(* IEC 61131-3 sources: Word/plc-course/10-structured-text/labs/solutions, 4 files *)

(* ---- 10-1-array-statistics.st ---- *)
(* Lab 10-1: Array statistics - ten cold-store temperature probes.
   Module 10 (Structured Text). REFERENCE SOLUTION - try the lab yourself first. *)

PROGRAM ArrayStats
  VAR (* interface: the I/O mapping routine copies the ten probe readings in here *)
    Samples  : ARRAY[1..10] OF REAL;  (* probe temperatures, degC. Samples[3] is probe TT-303 *)
    MinValue : REAL;                  (* coldest reading, degC *)
    MaxValue : REAL;                  (* warmest reading, degC *)
    Average  : REAL;                  (* mean of the ten readings, degC *)
    MaxIndex : INT;                   (* probe number (1..10) of the warmest reading *)
  END_VAR
  VAR CONSTANT
    NUM_PROBES : INT := 10;           (* must match the upper bound of Samples *)
  END_VAR
  VAR
    i   : INT;                        (* loop index *)
    Sum : REAL;                       (* running total, rebuilt from zero every scan *)
  END_VAR

  (* Start from the first sample, never from 0.0. In a freezer every reading is
     below zero, so a maximum that started at 0.0 would never be beaten. *)
  MinValue := Samples[1];
  MaxValue := Samples[1];
  MaxIndex := 1;
  Sum := 0.0;   (* Sum keeps its value between scans, so it must be cleared here *)

  FOR i := 1 TO NUM_PROBES DO
    Sum := Sum + Samples[i];

    IF Samples[i] < MinValue THEN
      MinValue := Samples[i];
    END_IF;

    (* Strictly greater: when two probes share the warmest value, the
       first one found (the lower probe number) is kept. *)
    IF Samples[i] > MaxValue THEN
      MaxValue := Samples[i];
      MaxIndex := i;
    END_IF;
  END_FOR;

  (* REAL division: both operands must be REAL, so convert the count. *)
  Average := Sum / INT_TO_REAL(NUM_PROBES);
END_PROGRAM

CONFIGURATION Config0
  RESOURCE Res0 ON PLC
    TASK MainTask(INTERVAL := T#10ms, PRIORITY := 0);
    PROGRAM Inst0 WITH MainTask : ArrayStats;
  END_RESOURCE
END_CONFIGURATION

(* ---- 10-2-median-filter.st ---- *)
(* Lab 10-2: Median filter for a noisy tank level.
   Module 10 (Structured Text). REFERENCE SOLUTION - try the lab yourself first. *)

PROGRAM MedianFilter
  VAR (* interface *)
    RawLevel      : REAL;   (* noisy level from the radar transmitter, % *)
    SampleTrig    : BOOL;   (* sample clock: each rising edge takes one sample *)
    FilteredLevel : REAL;   (* median of the last five samples, % *)
    Ready         : BOOL;   (* TRUE once five samples have been collected *)
  END_VAR
  VAR
    History    : ARRAY[1..5] OF REAL;  (* samples in arrival order: [1] oldest, [5] newest *)
    Sorted     : ARRAY[1..5] OF REAL;  (* working copy that gets sorted *)
    Count      : INT;                  (* samples collected so far, 0..5 *)
    SampleEdge : R_TRIG;               (* one sample per rising edge of SampleTrig *)
    i, j       : INT;
    Temp       : REAL;                 (* swap space for the sort *)
  END_VAR

  (* 1. Take a sample on each rising edge only. Holding SampleTrig TRUE for
        many scans must still give exactly one sample. *)
  SampleEdge(CLK := SampleTrig);
  IF SampleEdge.Q THEN
    (* Shift the history one place towards the old end. The oldest sample
       falls off, and the new one goes in at the newest end. *)
    FOR i := 1 TO 4 DO
      History[i] := History[i + 1];
    END_FOR;
    History[5] := RawLevel;
    IF Count < 5 THEN
      Count := Count + 1;
    END_IF;
  END_IF;

  Ready := Count >= 5;

  IF Ready THEN
    (* 2. Sort a COPY. The history must stay in time order, or the next shift
          would throw away the smallest value instead of the oldest one. *)
    Sorted := History;
    (* Bubble sort: each pass moves the largest remaining value to the end.
       Four passes are enough for five values (at most 10 comparisons). *)
    FOR i := 1 TO 4 DO
      FOR j := 1 TO 5 - i DO
        IF Sorted[j] > Sorted[j + 1] THEN
          Temp := Sorted[j];
          Sorted[j] := Sorted[j + 1];
          Sorted[j + 1] := Temp;
        END_IF;
      END_FOR;
    END_FOR;
    (* 3. The median of five sorted values is the middle one. *)
    FilteredLevel := Sorted[3];
  ELSE
    (* Warming up: pass the newest sample straight through, so the output is
       sensible from the first sample (it is 0.0 before any sample). *)
    FilteredLevel := History[5];
  END_IF;
END_PROGRAM

CONFIGURATION Config0
  RESOURCE Res0 ON PLC
    TASK MainTask(INTERVAL := T#10ms, PRIORITY := 0);
    PROGRAM Inst0 WITH MainTask : MedianFilter;
  END_RESOURCE
END_CONFIGURATION

(* ---- 10-3-strapping-table.st ---- *)
(* Lab 10-3: Tank strapping table - level to volume by piecewise-linear lookup.
   Module 10 (Structured Text). REFERENCE SOLUTION - try the lab yourself first. *)

(* Piecewise-linear interpolation in a table of 9 breakpoints.
   XTable must be strictly increasing. Outside the table the result is
   clamped to the first or last Y value and Clamped is set.

   The tables are VAR_IN_OUT, so they are passed by reference and not
   copied on every call. (MATIEC also cannot pass an array to a FUNCTION as
   a VAR_INPUT; CODESYS and TIA Portal can.) This function only reads them. *)
FUNCTION F_Interpolate : REAL
  VAR_IN_OUT
    XTable : ARRAY[1..9] OF REAL;   (* breakpoints, strictly increasing *)
    YTable : ARRAY[1..9] OF REAL;   (* value at each breakpoint *)
  END_VAR
  VAR_INPUT
    X : REAL;                       (* value to look up *)
  END_VAR
  VAR_OUTPUT
    Clamped : BOOL;                 (* TRUE when X is outside the table *)
  END_VAR
  VAR
    i    : INT;
    Span : REAL;
  END_VAR

  (* Guard clauses first: deal with the edge cases and leave early, so the
     main calculation below needs no extra nesting. *)
  Clamped := FALSE;
  IF X < XTable[1] THEN
    Clamped := TRUE;
    F_Interpolate := YTable[1];
    RETURN;
  END_IF;
  IF X > XTable[9] THEN
    Clamped := TRUE;
    F_Interpolate := YTable[9];
    RETURN;
  END_IF;

  (* Find the first segment whose upper breakpoint is at or above X.
     Segment i runs from XTable[i] to XTable[i + 1]. *)
  FOR i := 1 TO 8 DO
    IF X <= XTable[i + 1] THEN
      Span := XTable[i + 1] - XTable[i];
      IF Span > 0.0 THEN
        F_Interpolate := YTable[i] + (YTable[i + 1] - YTable[i]) * (X - XTable[i]) / Span;
      ELSE
        (* Two equal breakpoints: a typing error in the table. Avoid a
           division by zero and use the upper value. *)
        F_Interpolate := YTable[i + 1];
      END_IF;
      RETURN;   (* found it: later segments must not overwrite the result *)
    END_IF;
  END_FOR;

  (* Only reached if the table is not in increasing order. *)
  F_Interpolate := YTable[9];
END_FUNCTION

PROGRAM StrappingTable
  VAR (* interface *)
    Level      : REAL;   (* measured level, m (already scaled from the 4-20 mA signal) *)
    Volume     : REAL;   (* volume in the tank, m3 *)
    OutOfTable : BOOL;   (* TRUE when Level is below the first or above the last breakpoint *)
    (* Strapping table of a horizontal cylindrical tank, 2.0 m diameter and
       5.0 m long (15.708 m3 when full). The test may load other tables. *)
    LevelBP  : ARRAY[1..9] OF REAL := [0.0, 0.25, 0.5, 0.75, 1.0, 1.25, 1.5, 1.75, 2.0];
    VolumeBP : ARRAY[1..9] OF REAL := [0.0, 1.133, 3.071, 5.380, 7.854, 10.328, 12.637, 14.575, 15.708];
  END_VAR

  Volume := F_Interpolate(XTable := LevelBP, YTable := VolumeBP, X := Level,
                          Clamped => OutOfTable);
END_PROGRAM

CONFIGURATION Config0
  RESOURCE Res0 ON PLC
    TASK MainTask(INTERVAL := T#10ms, PRIORITY := 0);
    PROGRAM Inst0 WITH MainTask : StrappingTable;
  END_RESOURCE
END_CONFIGURATION

(* ---- 10-4-alarm-message.st ---- *)
(* Lab 10-4: Build an alarm message string for the operator.
   Module 10 (Structured Text). REFERENCE SOLUTION - try the lab yourself first. *)

PROGRAM AlarmMessage
  VAR (* interface *)
    TagName : STRING := 'TT-104';   (* instrument tag *)
    Units   : STRING := 'degC';     (* engineering units *)
    PV      : REAL;                 (* process value, -3000.0 .. 3000.0 *)
    HiHi    : BOOL;                 (* alarm states from the alarm logic *)
    Hi      : BOOL;
    Lo      : BOOL;
    LoLo    : BOOL;
    BadPV   : BOOL;                 (* signal fault: the value cannot be trusted *)
    Message : STRING;               (* text for the alarm banner, '' when healthy *)
  END_VAR
  VAR
    Tenths    : INT;      (* PV rounded to tenths: 87.46 -> 875 *)
    Sign      : STRING;   (* '-' or '' *)
    ValueText : STRING;   (* PV formatted with one decimal, e.g. '-0.4' *)
    StateText : STRING;   (* 'HIGH HIGH', 'HIGH', ... *)
  END_VAR

  (* 1. Format PV with exactly one decimal place.
        REAL_TO_STRING is no use here: MATIEC prints 87.4 as '87.40000153',
        and other platforms use other formats. Work in whole tenths instead. *)
  Tenths := REAL_TO_INT(PV * 10.0);      (* rounds to the nearest tenth *)
  IF Tenths < 0 THEN
    (* Take the sign off first. Otherwise -0.4 gives Tenths / 10 = 0 and the
       minus sign is lost, and MOD of a negative number is negative. *)
    Sign := '-';
    Tenths := -Tenths;
  ELSE
    Sign := '';                          (* -0.04 rounds to 0 and prints as 0.0 *)
  END_IF;
  ValueText := CONCAT(Sign, INT_TO_STRING(Tenths / 10), '.', INT_TO_STRING(Tenths MOD 10));

  (* 2. Choose the text for the most important active state. The order of the
        ELSIF chain IS the priority: the first TRUE condition wins. The
        trip-level alarms (HiHi, LoLo) come before the pre-alarms (Hi, Lo),
        because a latched low-low still matters more than a new high. *)
  IF BadPV THEN
    Message := CONCAT(TagName, ' BAD PV');   (* no value: it would be meaningless *)
  ELSE
    IF HiHi THEN
      StateText := 'HIGH HIGH';
    ELSIF LoLo THEN
      StateText := 'LOW LOW';
    ELSIF Hi THEN
      StateText := 'HIGH';
    ELSIF Lo THEN
      StateText := 'LOW';
    ELSE
      StateText := '';
    END_IF;

    IF StateText = '' THEN
      Message := '';                         (* healthy: clear the banner *)
    ELSE
      Message := CONCAT(TagName, ' ', StateText, ' ', ValueText, ' ', Units);
    END_IF;
  END_IF;
END_PROGRAM

CONFIGURATION Config0
  RESOURCE Res0 ON PLC
    TASK MainTask(INTERVAL := T#10ms, PRIORITY := 0);
    PROGRAM Inst0 WITH MainTask : AlarmMessage;
  END_RESOURCE
END_CONFIGURATION
